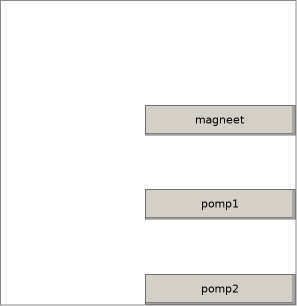
VISUALIZATION vKnoppen  // 297x306
    Button (145,105 150x30), "magneet", colour toggle: knoppen.bmagneet
        toggle knoppen.bmagneet
    Button (145,189 150x30), "pomp1", colour toggle: knoppen.bpomp1
        toggle knoppen.bpomp1
    Button (145,274 150x30), "pomp2", colour toggle: knoppen.bpomp2
        toggle knoppen.bpomp2
END_VISUALIZATION

(* stored: Version 1.1.0.1, ProductVersion 3.1.4024.2
   Visu vKnoppen: Id {2cab04fa-c71d-4c83-993a-af2c1a930aaf} *)
